// TIA Portal project "s05_pnname" (V21)

(* hardware
DEVICE "S7-1200 station_1"  S7-1200 Station
   slot 0: "Rack_0"  S7-1200 Rack  Rack  V1.0
   slot 1: "ZZALPHA"  CPU 1212C AC/DC/Rly  6ES7 212-1BD30-0XB0  V2.2
*)

// ===== PLC "ZZALPHA"  CPU 1212C AC/DC/Rly =====

ORGANIZATION_BLOCK "Main"   // OB1, LAD, ProgramCycle
TITLE = "Main Program Sweep (Cycle)"
{ S7_Optimized_Access := 'TRUE' }
VERSION : 0.1
BEGIN
END_ORGANIZATION_BLOCK